ABB RobotStudio station: ros2_srrc (IFRA-Cranfield) - IRB1200.rspag

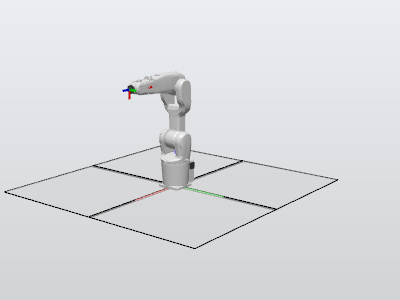
--- station ---
Station ros2_srrc (IFRA-Cranfield) - IRB1200 (saved by RobotStudio 22.3.10141.1)
Controller IRB1200_5_90
  mechanical unit ROB_1: IRB1200_5_90_STD_03, 6 joints, base frame (0, 0, 0) mm
Layout (positions relative to the parent item):
  - IRB1200_5_90_STD_03 [mechanism, from %ABB.RobotStudio.Models.IRB1200%\IRB1200_5_90_STD_03.rslib] at (0, 0, 0) mm; joint values [-0.0111, -0.0055, -0.0032, -0.001, 0.0066, -0.0054] (rad or m)

--- Controller Data/IRB1200_5_90/RAPID/TASK1/PROGMOD/TRob1Main.mod ---
MODULE TRob1Main
!======================================================================================================
! Copyright (c) 2018, ABB Schweiz AG
! All rights reserved.
!
! Redistribution and use in source and binary forms, with
! or without modification, are permitted provided that
! the following conditions are met:
!
!    * Redistributions of source code must retain the
!      above copyright notice, this list of conditions
!      and the following disclaimer.
!    * Redistributions in binary form must reproduce the
!      above copyright notice, this list of conditions
!      and the following disclaimer in the documentation
!      and/or other materials provided with the
!      distribution.
!    * Neither the name of ABB nor the names of its
!      contributors may be used to endorse or promote
!      products derived from this software without
!      specific prior wrSitten permission.
!
! THIS SOFTWARE IS PROVIDED BY THE COPYRIGHT HOLDERS AND CONTRIBUTORS "AS IS"
! AND ANY EXPRESS OR IMPLIED WARRANTIES, INCLUDING, BUT NOT LIMITED TO, THE
! IMPLIED WARRANTIES OF MERCHANTABILITY AND FITNESS FOR A PARTICULAR PURPOSE
! ARE DISCLAIMED. IN NO EVENT SHALL THE COPYRIGHT HOLDER OR CONTRIBUTORS BE
! LIABLE FOR ANY DIRECT, INDIRECT, INCIDENTAL, SPECIAL, EXEMPLARY, OR CONSEQUENTIAL
! DAMAGES (INCLUDING, BUT NOT LIMITED TO, PROCUREMENT OF SUBSTITUTE GOODS OR
! SERVICES; LOSS OF USE, DATA, OR PROFITS; OR BUSINESS INTERRUPTION) HOWEVER
! CAUSED AND ON ANY THEORY OF LIABILITY, WHETHER IN CONTRACT, STRICT LIABILITY,
! OR TORT (INCLUDING NEGLIGENCE OR OTHERWISE) ARISING IN ANY WAY OUT OF THE USE OF
! THIS SOFTWARE, EVEN IF ADVISED OF THE POSSIBILITY OF SUCH DAMAGE.
!======================================================================================================

!======================================================================================================
! Copyright (c) 2023, IFRA-Cranfield - Cranfield University, UK.
!
!   IFRA (Intelligent Flexible Robotics and Assembly) Group, CRANFIELD UNIVERSITY
!   Created on behalf of the IFRA Group at Cranfield University, United Kingdom
!   E-mail: IFRA@cranfield.ac.uk
!
!   The TRob1Main.mod file provided in the public abb_ros2 (https://github.com/PickNikRobotics/abb_ros2)
!   GitHub repository has been modified, obtaining better results and an improved Robot Motion.
!   The ROS2-Control of the ABB IRB120 robot is realised through the ros2srrc_irb120_bringup ROS2 package,
!   which is publicly available in the ros2_SimRealRobotControl GitHub repository:
!         * https://github.com/IFRA-Cranfield/ros2_SimRealRobotControl
!
!   AUTHORS:
!     - Mikel Bueno Viso - Mikel.Bueno-Viso@cranfield.ac.uk
!     - Dr. Seemal Asif - s.asif@cranfield.ac.uk
!     - Prof. Phil Webb - p.f.webb@cranfield.ac.uk
!
!   DATE: April, 2023.
!
!======================================================================================================

    !***********************************************************
    ! Program data
    !***********************************************************
    ! Home position.
    LOCAL CONST jointtarget home := [[0, 0, 0, 0, 30, 0], [9E9, 9E9, 9E9, 9E9, 9E9, 9E9]];

    ! Identifier for the EGM correction.
    LOCAL VAR egmident egm_id;

    ! Limits for convergance.
    LOCAL VAR egm_minmax egm_condition := [-0.1, 0.1];
    LOCAL VAR egm_minmax egm_condition_lin := [-1, 1];

    !***********************************************************
    !
    ! Procedure main
    !
    !   This RAPID code exemplify how to run EGM joint position
    !   motions.
    !
    !   Note: Update the UCDevice "ROB_1" with correct
    !         values for the remote address and port
    !         (i.e. to the EGM server).
    !
    !         Update via RobotStudio:
    !         Controller tab -> Configuration ->
    !         Communication -> Transmission Protocol
    !
    !***********************************************************
    PROC main()
        MoveAbsJ home, v200, fine, tool0;


        ! Register an EGM id.
        EGMGetId egm_id;

        ! Setup the EGM communication.
        EGMSetupUC ROB_1, egm_id, "default", "ROB_1", \Joint;

        ! Prepare for an EGM communication session.
        EGMActJoint egm_id
                    \J1:=egm_condition
                    \J2:=egm_condition
                    \J3:=egm_condition
                    \J4:=egm_condition
                    \J5:=egm_condition
                    \J6:=egm_condition
                    \LpFilter:=20
                    \SampleRate:=4
                    \MaxPosDeviation:=2000
                    \MaxSpeedDeviation:=250.0;
        WHILE TRUE DO
            ! Start the EGM communication session.
            EGMRunJoint egm_id, EGM_STOP_HOLD, \J1 \J2 \J3 \J4 \J5 \J6 \CondTime:=1 \RampOutTime:=1 \PosCorrGain:=0;
        ENDWHILE
        ! Release the EGM id.
        EGMReset egm_id;


    ERROR
        IF ERRNO = ERR_UDPUC_COMM THEN
            TPWrite "Communication timedout";
            TRYNEXT;
        ENDIF
    ENDPROC
ENDMODULE
